// TIA Portal V18 export
FUNCTION_BLOCK "BO_Torq"   // FB33, LAD
TITLE = Break Out
{ S7_Optimized_Access := 'TRUE' }
// Written BY Kristopher Gimenez Feb 7,2023
// This block is used to control the TD Break Out Torq mode
// stored: AutoNumber false, MemoryReserve 100, SetENOAutomatically false
   VAR_INPUT
      Start : Bool;
   END_VAR
   VAR_OUTPUT
      FlowRevmAOut : Real;
      EnableP1 : Bool;
      EnableP2 { ExternalWritable := 'False'} : Bool;
      BOEn : Bool;
      BOSeqRunning : Bool;
   END_VAR
   VAR
      PumpToggle : Bool;   // Bit will toggle each make up sequence to choose which pump to stroke. 0 = P1, 1 = P2, TBD if using this in BO.
      RampDown : Bool;   // Bit to know system need to ramp down
      RampDownComplete : Bool;   // Indicates Ramp Down completed
      Flow_Ramp { S7_SetPoint := 'True'} : RampFunction;
      FlowRampInmA : Real;   // Value assigned to ramp fucntion to get ramped ouput
      BOFlowmA : Real;
      BOSeqRunLast : Bool;
   END_VAR
   VAR_TEMP
      tempReal : Real;
      toggleTemp : Bool;
   END_VAR
BEGIN

REGION Network 1: Set Running
   // Set running bit and trigger resets when starting a MU sequence
   // Pump Toggle is set but may not be needed for BO mode
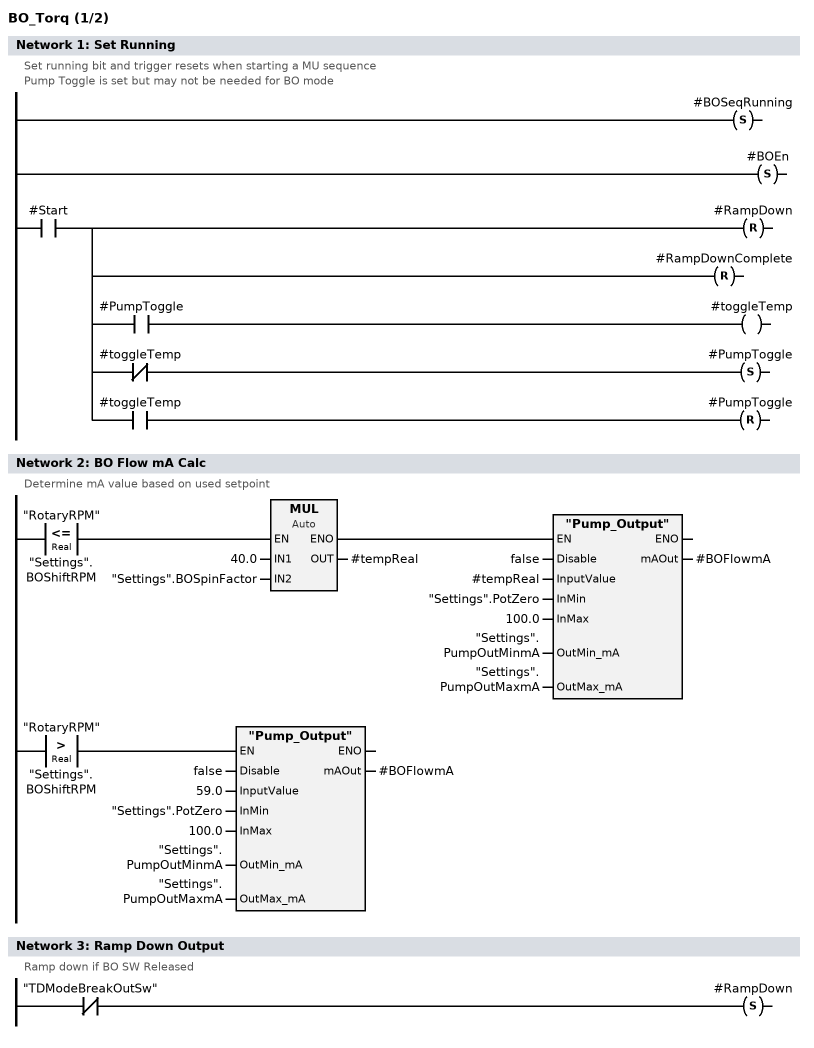
   RUNG wire#powerrail
      S_Coil( #BOSeqRunning )
   END_RUNG
   RUNG wire#powerrail
      S_Coil( #BOEn )
   END_RUNG
   RUNG wire#powerrail
      Contact( #Start )
      wire#w1
      R_Coil( #RampDown )
   END_RUNG
   RUNG wire#w1
      R_Coil( #RampDownComplete )
   END_RUNG
   RUNG wire#w1
      Contact( #PumpToggle )
      Coil( #toggleTemp )
   END_RUNG
   RUNG wire#w1
      I_Contact( #toggleTemp )
      S_Coil( #PumpToggle )
   END_RUNG
   RUNG wire#w1
      Contact( #toggleTemp )
      R_Coil( #PumpToggle )
   END_RUNG
   // the same network as SCL:
   #BOSeqRunning := TRUE;
   #BOEn := TRUE;
   IF #Start THEN
       #RampDown := FALSE;
       #RampDownComplete := FALSE;
   END_IF;
   #toggleTemp := #Start AND #PumpToggle;
   IF #Start AND NOT #toggleTemp THEN #PumpToggle := TRUE; END_IF;
   IF #Start AND #toggleTemp THEN #PumpToggle := FALSE; END_IF;
END_REGION

REGION Network 2: BO Flow mA Calc
   // Determine mA value based on used setpoint
   RUNG wire#powerrail
      { S7_Templates := "SrcType := Real" } LE_Contact(in1 := "RotaryRPM", in2 := "Settings".BOShiftRPM)
      Mul(in1 := 40.0, in2 := "Settings".BOSpinFactor, out => #tempReal)
      "Pump_Output"(Disable := false, InputValue := #tempReal, InMin := "Settings".PotZero, InMax := 100.0, OutMin_mA := "Settings".PumpOutMinmA, OutMax_mA := "Settings".PumpOutMaxmA, mAOut => #BOFlowmA)
   END_RUNG
   RUNG wire#powerrail
      { S7_Templates := "SrcType := Real" } GT_Contact(in1 := "RotaryRPM", in2 := "Settings".BOShiftRPM)
      "Pump_Output"(Disable := false, InputValue := 59.0, InMin := "Settings".PotZero, InMax := 100.0, OutMin_mA := "Settings".PumpOutMinmA, OutMax_mA := "Settings".PumpOutMaxmA, mAOut => #BOFlowmA)
   END_RUNG
   // the same network as SCL:
   IF "RotaryRPM" <= "Settings".BOShiftRPM THEN
       #tempReal := 40.0 * "Settings".BOSpinFactor;
       "Pump_Output"(Disable := false,
                     InputValue := #tempReal,
                     InMin := "Settings".PotZero,
                     InMax := 100.0,
                     OutMin_mA := "Settings".PumpOutMinmA,
                     OutMax_mA := "Settings".PumpOutMaxmA,
                     mAOut => #BOFlowmA);
   END_IF;
   IF "RotaryRPM" > "Settings".BOShiftRPM THEN
       "Pump_Output"(Disable := false,
                     InputValue := 59.0,
                     InMin := "Settings".PotZero,
                     InMax := 100.0,
                     OutMin_mA := "Settings".PumpOutMinmA,
                     OutMax_mA := "Settings".PumpOutMaxmA,
                     mAOut => #BOFlowmA);
   END_IF;
END_REGION

REGION Network 3: Ramp Down Output
   // Ramp down if BO SW Released
   RUNG wire#powerrail
      I_Contact( "TDModeBreakOutSw" )
      S_Coil( #RampDown )
   END_RUNG
   // the same network as SCL:
   IF NOT "TDModeBreakOutSw" THEN #RampDown := TRUE; END_IF;
END_REGION

REGION Network 4: Assign Flow Ramp Parameters
   // Set Flow Ramp settings as needed. Note no changes to flow ramp in various Auto MU ranges.
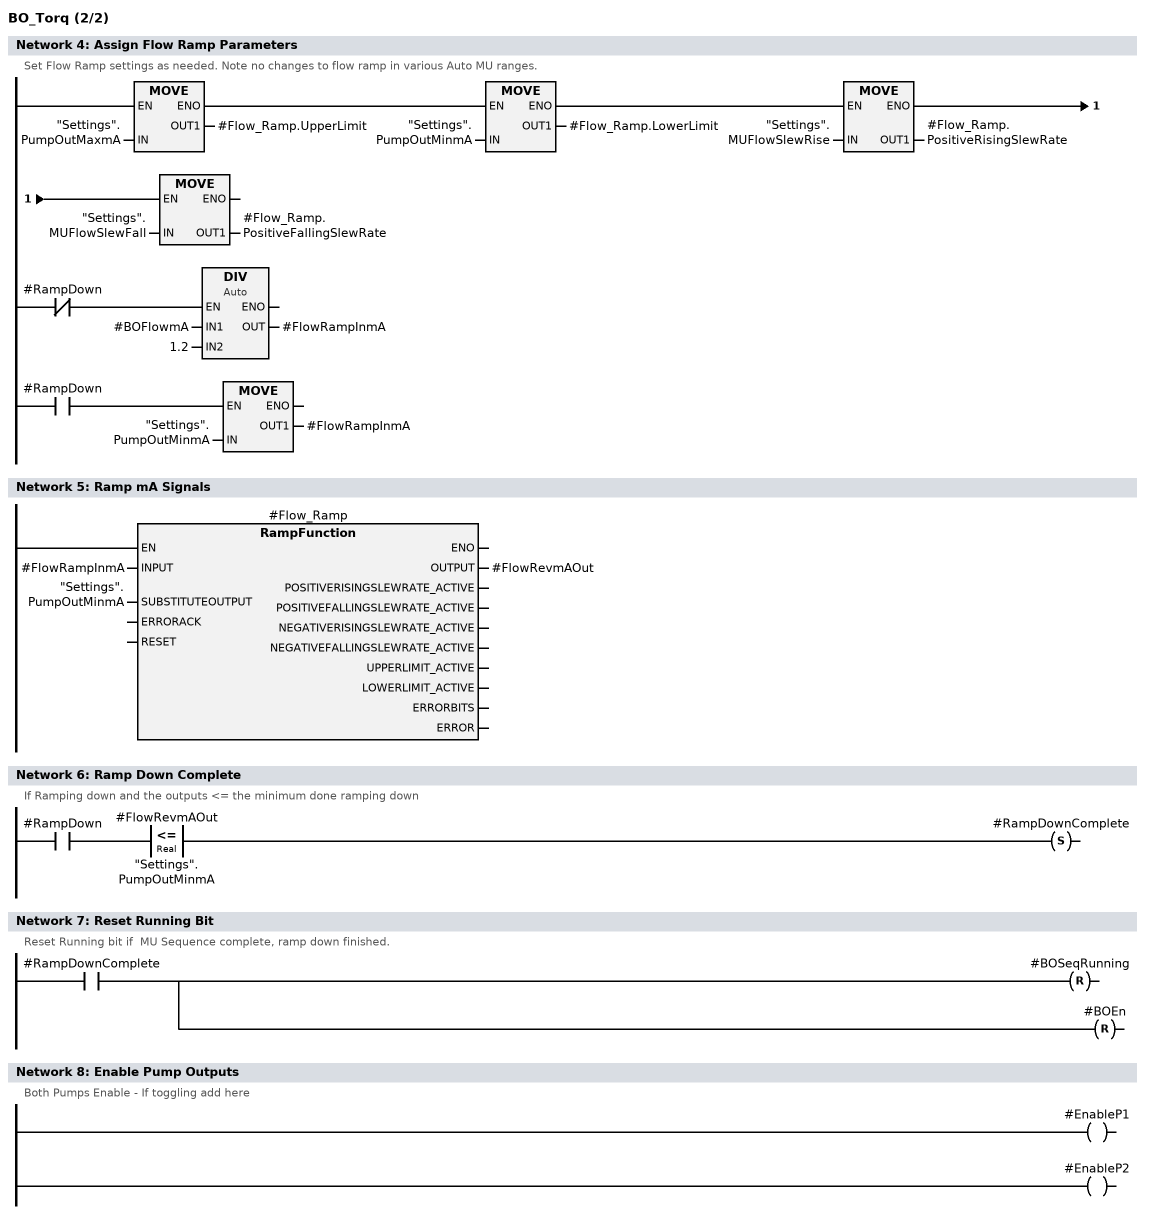
   RUNG wire#powerrail
      Move(in := "Settings".PumpOutMaxmA, out1 => #Flow_Ramp.UpperLimit)
      Move(in := "Settings".PumpOutMinmA, out1 => #Flow_Ramp.LowerLimit)
      Move(in := "Settings".MUFlowSlewRise, out1 => #Flow_Ramp.PositiveRisingSlewRate)
      Move(in := "Settings".MUFlowSlewFall, out1 => #Flow_Ramp.PositiveFallingSlewRate)
   END_RUNG
   RUNG wire#powerrail
      I_Contact( #RampDown )
      Div(in1 := #BOFlowmA, in2 := 1.2, out => #FlowRampInmA)
   END_RUNG
   RUNG wire#powerrail
      Contact( #RampDown )
      Move(in := "Settings".PumpOutMinmA, out1 => #FlowRampInmA)
   END_RUNG
   // the same network as SCL:
   #Flow_Ramp.UpperLimit := "Settings".PumpOutMaxmA;
   #Flow_Ramp.LowerLimit := "Settings".PumpOutMinmA;
   #Flow_Ramp.PositiveRisingSlewRate := "Settings".MUFlowSlewRise;
   #Flow_Ramp.PositiveFallingSlewRate := "Settings".MUFlowSlewFall;
   IF NOT #RampDown THEN #FlowRampInmA := #BOFlowmA / 1.2; END_IF;
   IF #RampDown THEN #FlowRampInmA := "Settings".PumpOutMinmA; END_IF;
END_REGION

REGION Network 5: Ramp mA Signals
   RUNG wire#powerrail
      #Flow_Ramp.RampFunction(Input := #FlowRampInmA, SubstituteOutput := "Settings".PumpOutMinmA, ErrorAck :=, Reset :=, Output => #FlowRevmAOut, PositiveRisingSlewRate_Active =>, PositiveFallingSlewRate_Active =>, NegativeRisingSlewRate_Active =>, NegativeFallingSlewRate_Active =>, UpperLimit_Active =>, LowerLimit_Active =>, ErrorBits =>, Error =>)
   END_RUNG
   // the same network as SCL:
   #Flow_Ramp(Input := #FlowRampInmA, SubstituteOutput := "Settings".PumpOutMinmA, Output => #FlowRevmAOut);   // RampFunction
END_REGION

REGION Network 6: Ramp Down Complete
   // If Ramping down and the outputs <= the minimum done ramping down
   RUNG wire#powerrail
      Contact( #RampDown )
      { S7_Templates := "SrcType := Real" } LE_Contact(in1 := #FlowRevmAOut, in2 := "Settings".PumpOutMinmA)
      S_Coil( #RampDownComplete )
   END_RUNG
   // the same network as SCL:
   IF #RampDown AND (#FlowRevmAOut <= "Settings".PumpOutMinmA) THEN #RampDownComplete := TRUE; END_IF;
END_REGION

REGION Network 7: Reset Running Bit
   // Reset Running bit if  MU Sequence complete, ramp down finished.
   RUNG wire#powerrail
      Contact( #RampDownComplete )
      wire#w1
      R_Coil( #BOSeqRunning )
   END_RUNG
   RUNG wire#w1
      R_Coil( #BOEn )
   END_RUNG
   // the same network as SCL:
   IF #RampDownComplete THEN
       #BOSeqRunning := FALSE;
       #BOEn := FALSE;
   END_IF;
END_REGION

REGION Network 8: Enable Pump Outputs
   // Both Pumps Enable - If toggling add here
   RUNG wire#powerrail
      Coil( #EnableP1 )
   END_RUNG
   RUNG wire#powerrail
      Coil( #EnableP2 )
   END_RUNG
   // the same network as SCL:
   #EnableP1 := TRUE;
   #EnableP2 := TRUE;
END_REGION
END_FUNCTION_BLOCK
